ABB RobotStudio station: TPL1.rsstnx

Station TPL1 (saved by RobotStudio 25.5.11605.0)
Controller IRB140_6_81
  mechanical unit ROB_1: IRB140_6_81_C_03, 6 joints, base frame (0, 0, 0) mm
Layout (positions relative to the parent item):
  - IRB140_6_81_C_03 [mechanism, from %ABB.RobotStudio.Models.IRB140%\IRB140_6_81_C_G_03.rslib] at (0, 0, 0) mm; joint values [-0.0715, -0.0782, 0.0753, 0.1225, 0.5309, -0.1415] (rad or m)
  - Mesa [part], size 365 x 405 x 340 mm
  - Perno [part], size 20 x 100 x 20 mm
  - Pinza [mechanism] at (477.09, -30.13, 679.5) mm, rotated rx 180 ry 60 rz 180 deg
      TCP Pinza at (0, 0, 137) mm, rotated rx 0 ry 0 rz -22.5 deg
      links: Dummy
Attachment: Pinza is attached to IRB140_6_81_C_03 / Link6
Collision set Conjunto de colisión_1: Mesa against Perno, near miss 0.02 m
EventTableEntry 2467: ActivationMode=2, Cyclic=false, Group=, Trigger=DO_Pinza 2468, Actions=[EventTableActionAttach 2469], Comment=
EventTableTriggerIO 2468: Operator=0, IOValue=[1], IRC5Controller=? -1, SignalSource=IRB140_6_81 1261
EventTableActionAttach 2469: MountObject=false, FlangeIndext=0, FindNearest=false, AttachmentParent=Pinza 2362, AttachmentChild=Perno 2358, Offset=[X=1, Y=0, Z=0, W=0, X=0, Y=1, Z=0, W=0, X=0, Y=0, Z=1, W=0, X=0, Y=0, Z=0, W=1]
EventTableEntry 2470: ActivationMode=2, Cyclic=false, Group=, Trigger=DO_Pinza 2471, Actions=[EventTableActionDetach 2472], Comment=
EventTableTriggerIO 2471: Operator=0, IOValue=[0], IRC5Controller=? -1, SignalSource=IRB140_6_81 1261
EventTableActionDetach 2472: AttachmentParent=Pinza 2362, AttachmentChild=Perno 2358
Targets, tools, work objects and paths stored in the station, written as RAPID:
! task T_ROB1
MODULE CalibData
  PERS tooldata Pinza:=[TRUE,[[0,0,137],[0.980785,0,0,-0.19509]],[0.5,[0,0,100],[1,0,0,0],0,0,0]];
  PERS wobjdata Agujero_woj:=[FALSE,TRUE,"",[[600,-60,260],[1,0,0,0]],[[0,0,0],[1,0,0,0]]];
  PERS wobjdata perno_woj:=[FALSE,TRUE,"",[[400,180,130],[1,0,0,0]],[[0,0,0],[1,0,0,0]]];
ENDMODULE

! task T_ROB1
MODULE Module1
  CONST robtarget agujero_t:=[[0,0,0],[0,0,1,0],[0,0,0,0],[9E+09,9E+09,9E+09,9E+09,9E+09,9E+09]];
  CONST robtarget perno_t:=[[0,0,0],[0.707106781,0.707106781,0,0],[0,0,0,0],[9E+09,9E+09,9E+09,9E+09,9E+09,9E+09]];
  CONST robtarget home_t:=[[624,0,611],[0.49039264,-0.168953175,0.849384968,-0.097545161],[0,0,0,0],[9E+09,9E+09,9E+09,9E+09,9E+09,9E+09]];
  CONST robtarget perno_alejado2:=[[100,-50,200],[0,1,0,0],[0,0,-2,0],[9E+09,9E+09,9E+09,9E+09,9E+09,9E+09]];
  CONST robtarget perno_t_vertical:=[[0,0,0],[0.707106781,0.707106781,0,0],[0,0,0,0],[9E+09,9E+09,9E+09,9E+09,9E+09,9E+09]];
  PROC main()
    AbrirPinza;
    Home;
    Trayecto_vertical;
    Home;
  ENDPROC
  PROC ColocarPerno()
    MoveJ perno_alejado2,V500,z50,Pinza\WObj:=perno_woj;
    MoveJ Offs(agujero_t,0,0,long_perno+aprox_agujero),v1000,z100,Pinza\WObj:=Agujero_woj;
    MoveL Offs(agujero_t,0,0,long_perno-prof_penetracion_agujero),v50,fine,Pinza\WObj:=Agujero_woj;
    AbrirPinza;
  ENDPROC
  PROC Home()
    MoveJ home_t,v100,z50,Pinza;
  ENDPROC
  PROC AbrirPinza()
    SetDO DO_Pinza,0;
    WaitTime 0.2;
  ENDPROC
  PROC CerrarPinza()
    SetDO DO_Pinza,1;
    WaitTime 0.2;
  ENDPROC
  PROC Trayecto_horizontal()
    ColocarPerno;
  ENDPROC
  PROC Trayecto_vertical()
    ColocarPerno;
  ENDPROC
ENDMODULE

